FUNCTION_BLOCK T_ComponentsCollection EXTENDS T_CollectionBase IMPLEMENTS I_ComponentsCollection

METHOD PUBLIC AddComponent : BOOL
VAR_INPUT
  newComponent : I_ComponentBase;
END_VAR
VAR
	item : I_InterfaceBase;
END_VAR
IF newComponent = 0 THEN
	LogError( 'Cannot AddComponent invalid ref' );
	RETURN;
END_IF

IF NOT __QUERYINTERFACE(newComponent, item) THEN
	LogError( 'Cannot AddComponent  NOT __QUERYINTERFACE(newComponent, item)' );
	RETURN;
END_IF

IF HasItem( item := item ) THEN
	LogWarning( 'Component already in collection.' );
	RETURN;
END_IF

AddComponent := addInSpareSlot( item := item );
END_METHOD

//! @summary Sets permissive bit to allow HMI control of component functions
METHOD PUBLIC AllowHMIControl
//! @description This method is called as required by the parent module of this component
VAR
	i : UDINT;
	Component : I_ComponentBase;
	item : I_InterfaceBase;
END_VAR
IF Count = 0 THEN
  RETURN;
END_IF

FOR i := 0 TO Count -1 DO

	IF NOT 	TryGetItem(i, item => item) THEN
		RETURN;
	END_IF
	
	IF NOT __QUERYINTERFACE(item, component) THEN
		RETURN;
	END_IF
		
	Component.AllowHMIControl();
		
END_FOR
END_METHOD

PROPERTY PUBLIC AnyError : BOOL
GET
VAR
  i : UDINT;
  Component : I_ComponentBase;
  item : I_InterfaceBase;
END_VAR
IF Count = 0 THEN
  RETURN;
END_IF

FOR i := 0 TO Count -1 DO

	IF NOT 	TryGetItem(i, item => item) THEN
		RETURN;
	END_IF
	
	IF NOT __QUERYINTERFACE(item, component) THEN
		RETURN;
	END_IF
		
	IF Component.Error THEN
		AnyError := TRUE;
		RETURN;
	END_IF

END_FOR
END_GET
END_PROPERTY

//! @summary Clears permissive bit to allow HMI control of component functions
METHOD PUBLIC BlockHMIControl
//! @description This method is called as required by the parent module of this component
VAR
	i : UDINT;
	Component : I_ComponentBase;
	item : I_InterfaceBase;
END_VAR
IF Count = 0 THEN
  RETURN;
END_IF

FOR i := 0 TO Count -1 DO

	IF NOT 	TryGetItem(i, item => item) THEN
		RETURN;
	END_IF
	
	IF NOT __QUERYINTERFACE(item, component) THEN
		RETURN;
	END_IF
		
	Component.BlockHMIControl();
		
END_FOR
END_METHOD

METHOD CyclicLogic
VAR
  i : UDINT;
  Component : I_ComponentBase;
  item : I_InterfaceBase;
END_VAR
IF Count = 0 THEN
  RETURN;
END_IF

FOR i := 0 TO Count -1 DO
	TryGetItem(i, item => item);
	__QUERYINTERFACE(item, component);
	IF component <> 0 THEN
  		Component.CyclicLogic();
	END_IF	
END_FOR
END_METHOD

PROPERTY PUBLIC InitialisedAll : BOOL
GET
VAR
  i : UDINT;
  Component : I_ComponentBase;
  item : I_InterfaceBase;
 END_VAR
IF Count = 0 THEN
	InitialisedAll := TRUE;
  RETURN;
END_IF

FOR i := 0 TO Count -1 DO

	IF NOT 	TryGetItem(i, item => item) THEN
		RETURN;
	END_IF
	
	IF NOT __QUERYINTERFACE(item, component) THEN
		RETURN;
	END_IF
		
	IF NOT Component.InitComplete THEN
		RETURN;
	END_IF
		

END_FOR

InitialisedAll := TRUE;
END_GET
END_PROPERTY

METHOD PUBLIC Reset
VAR
	i : UDINT;
	Component : I_ComponentBase;
	item : I_InterfaceBase;
END_VAR
IF Count = 0 THEN
  RETURN;
END_IF

FOR i := 0 TO Count -1 DO

	IF NOT 	TryGetItem(i, item => item) THEN
		RETURN;
	END_IF
	
	IF NOT __QUERYINTERFACE(item, component) THEN
		RETURN;
	END_IF
		
	Component.Reset();
		
END_FOR
END_METHOD

METHOD TryGetComponent: BOOL
VAR_INPUT
	index : UDINT;
END_VAR
VAR_OUTPUT
	component : I_ComponentBase;
END_VAR
VAR
	item : I_InterfaceBase;
END_VAR
IF NOT SUPER^.TryGetItem(index := index, item => item) THEN
	LogError( 'Cannot TryGetComponent NOT SUPER^.TryGetItem(index := index, item => item) ' );
	RETURN;
END_IF

IF NOT __QUERYINTERFACE(item, component) THEN
	LogError( 'Cannot TryGetComponent   NOT __QUERYINTERFACE(item, component) ' );
	RETURN;
END_IF

TryGetComponent := component <> 0;
END_METHOD

END_FUNCTION_BLOCK

(* stored: Version 1.1.0.1, ProductVersion 3.1.4024.12
   POU T_ComponentsCollection: Id {d0fd4ea2-8a96-0365-36ba-9fa85df78835}, SpecialFunc None
   Method AddComponent: Id {fb6c4003-1a4c-0530-3ee6-4677519bc680}
   Method AllowHMIControl: Id {a3a8d4ad-9d48-4f3f-ba31-3be39f8e4d90}
   Property AnyError: Id {9034e9d6-c017-4e85-8fb5-b86ce3eee340}
   Get Get: Id {9bb5938c-c9cb-4e41-99b0-44351b5c2d05}
   Method BlockHMIControl: Id {6f9e39dd-3470-4035-afab-a0932af02961}
   Method CyclicLogic: Id {91fecff3-afbd-4edb-b80e-debfd3f550ae}
   Property InitialisedAll: Id {c45efdcd-ff68-4ada-b178-9f283cfc29ff}
   Get Get: Id {b0c84a63-02dc-419d-8b39-3ee695183c82}
   Method Reset: Id {a96c8941-de5e-4d1c-bfc5-4f208123d152}
   Method TryGetComponent: Id {2d1e8721-47b6-026d-04e2-daccf35cf2e5} *)
